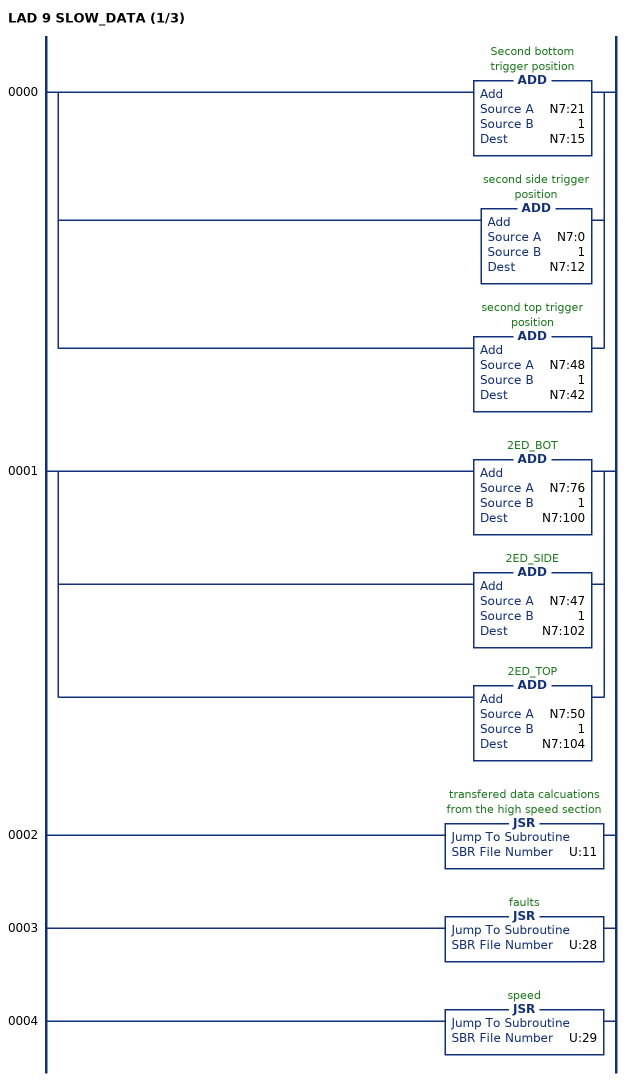
% Rung: 0 %
SOR BST ADD N7:21 1 N7:15 NXB ADD N7:0 1 N7:12 NXB ADD N7:48 1 N7:42 BND EOR
%   N7:21  BOT_TRIG_POS_INTEGER  "Trigger Position" %
%   N7:15  "Second bottom trigger position" %
%   N7:0  SIDE_TRIG_POS_INTEGE  "Side Trigger Position" %
%   N7:12  "second side trigger position" %
%   N7:48  TOP_TRIG_POS_INTEGER  "Top Trigger Position" %
%   N7:42  "second top trigger position" %
% Rung: 1 %
SOR BST ADD N7:76 1 N7:100 NXB ADD N7:47 1 N7:102 NXB ADD N7:50 1 N7:104 BND EOR
%   N7:76  BOT_TEST_LOC  "Location of pass window." %
%   N7:100  2ED_BOT %
%   N7:47  SIDE_TEST_LOC  "Location of pass window" %
%   N7:102  2ED_SIDE %
%   N7:50  TOP_TEST_LOC  "Location of pass window" %
%   N7:104  2ED_TOP %
% Rung: 2 %
SOR JSR U:11 EOR
%   U:11  "transfered data calcuations from the high speed section" %
% Rung: 3 %
SOR JSR U:28 EOR
%   U:28  "faults" %
% Rung: 4 %
SOR JSR U:29 EOR
%   U:29  "speed" %

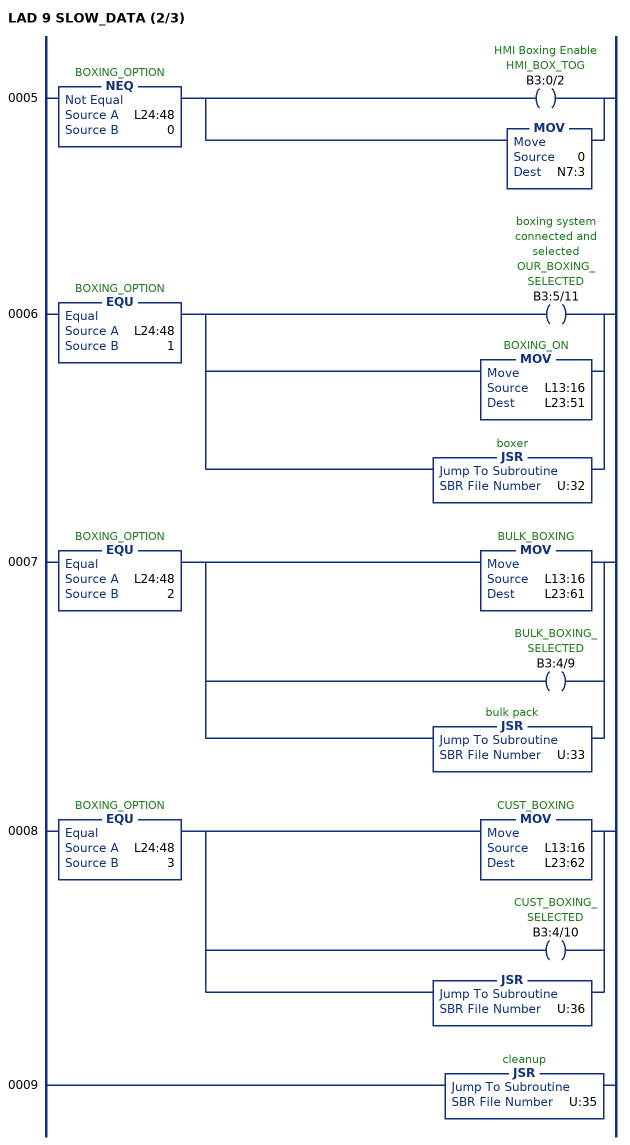
% Rung: 5 %
SOR NEQ L24:48 0 BST OTE B3:0/2 NXB MOV 0 N7:3 BND EOR
%   L24:48  BOXING_OPTION %
%   B3:0/2  HMI_BOX_TOG  "HMI Boxing Enable" %
% Rung: 6 %
SOR EQU L24:48 1 BST OTE B3:5/11 NXB MOV L13:16 L23:51 NXB JSR U:32 BND EOR
%   L24:48  BOXING_OPTION %
%   B3:5/11  OUR_BOXING_SELECTED  "boxing system connected and selected" %
%   L13:16  TRUE  "ONE TIME ENABLE FOR THE TIMES WHEN WE FORGET TO RE-ENABLE AFTER SHIPMENT" %
%   L23:51  BOXING_ON %
%   U:32  "boxer" %
% Rung: 7 %
SOR EQU L24:48 2 BST MOV L13:16 L23:61 NXB OTE B3:4/9 NXB JSR U:33 BND EOR
%   L24:48  BOXING_OPTION %
%   L13:16  TRUE  "ONE TIME ENABLE FOR THE TIMES WHEN WE FORGET TO RE-ENABLE AFTER SHIPMENT" %
%   L23:61  BULK_BOXING %
%   B3:4/9  BULK_BOXING_SELECTED %
%   U:33  "bulk pack" %
% Rung: 8 %
SOR EQU L24:48 3 BST MOV L13:16 L23:62 NXB OTE B3:4/10 NXB JSR U:36 BND EOR
%   L24:48  BOXING_OPTION %
%   L13:16  TRUE  "ONE TIME ENABLE FOR THE TIMES WHEN WE FORGET TO RE-ENABLE AFTER SHIPMENT" %
%   L23:62  CUST_BOXING %
%   B3:4/10  CUST_BOXING_SELECTED %
% Rung: 9 %
SOR JSR U:35 EOR
%   U:35  "cleanup" %

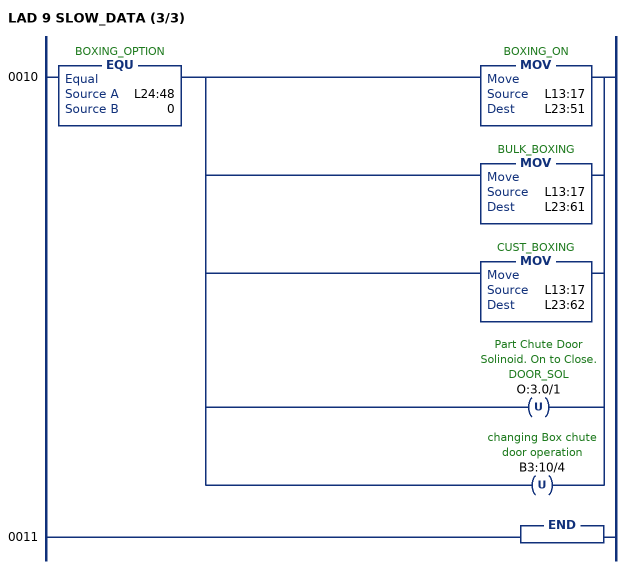
% Rung: 10 %
SOR EQU L24:48 0 BST MOV L13:17 L23:51 NXB MOV L13:17 L23:61 NXB MOV L13:17 L23:62 NXB OTU O:3.0/1 NXB OTU B3:10/4 BND EOR
%   L24:48  BOXING_OPTION %
%   L13:17  FALSE %
%   L23:51  BOXING_ON %
%   L23:61  BULK_BOXING %
%   L23:62  CUST_BOXING %
%   O:3.0/1  DOOR_SOL  "Part Chute Door Solinoid. On to Close." %
%   B3:10/4  "changing Box chute door operation" %
% Rung: 11 %
SOR END EOR

LADDER 10 "BOT_NUT"
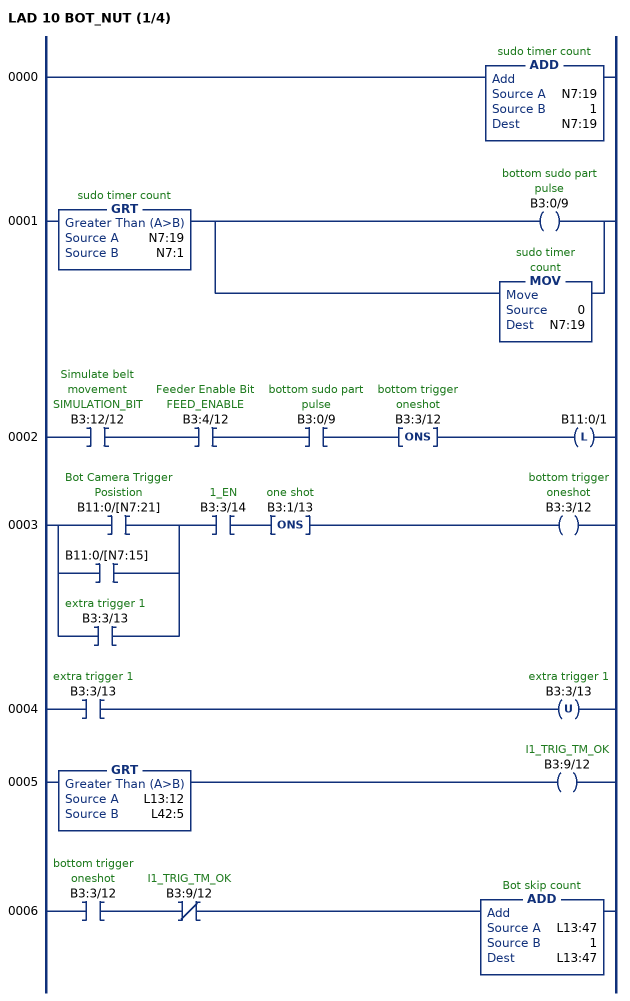
% Rung: 0 %
SOR ADD N7:19 1 N7:19 EOR
%   N7:19  "sudo timer count" %
% Rung: 1 %
SOR GRT N7:19 N7:1 BST OTE B3:0/9 NXB MOV 0 N7:19 BND EOR
%   N7:19  "sudo timer count" %
%   N7:1  "sudo part interval" %
%   B3:0/9  "bottom sudo part pulse" %
% Rung: 2 %
SOR XIC B3:12/12 XIC B3:4/12 XIC B3:0/9 ONS B3:3/12 OTL B11:0/1 EOR
%   B3:12/12  SIMULATION_BIT  "Simulate belt movement" %
%   B3:4/12  FEED_ENABLE  "Feeder Enable Bit" %
%   B3:0/9  "bottom sudo part pulse" %
%   B3:3/12  "bottom trigger oneshot" %
% Rung: 3 %
SOR BST XIC B11:0/[N7:21] NXB XIC B11:0/[N7:15] NXB XIC B3:3/13 BND XIC B3:3/14 ONS B3:1/13 OTE B3:3/12 EOR
%   B11:0/[N7:21]  "Bot Camera Trigger Posistion" %
%   N7:21  BOT_TRIG_POS_INTEGER  "Trigger Position" %
%   N7:15  "Second bottom trigger position" %
%   B3:3/13  "extra trigger 1" %
%   B3:3/14  1_EN %
%   B3:1/13  "one shot" %
%   B3:3/12  "bottom trigger oneshot" %
% Rung: 4 %
SOR XIC B3:3/13 OTU B3:3/13 EOR
%   B3:3/13  "extra trigger 1" %
% Rung: 5 %
SOR GRT L13:12 L42:5 OTE B3:9/12 EOR
%   B3:9/12  I1_TRIG_TM_OK %
% Rung: 6 %
SOR XIC B3:3/12 XIO B3:9/12 ADD L13:47 1 L13:47 EOR
%   B3:3/12  "bottom trigger oneshot" %
%   B3:9/12  I1_TRIG_TM_OK %
%   L13:47  "Bot skip count" %

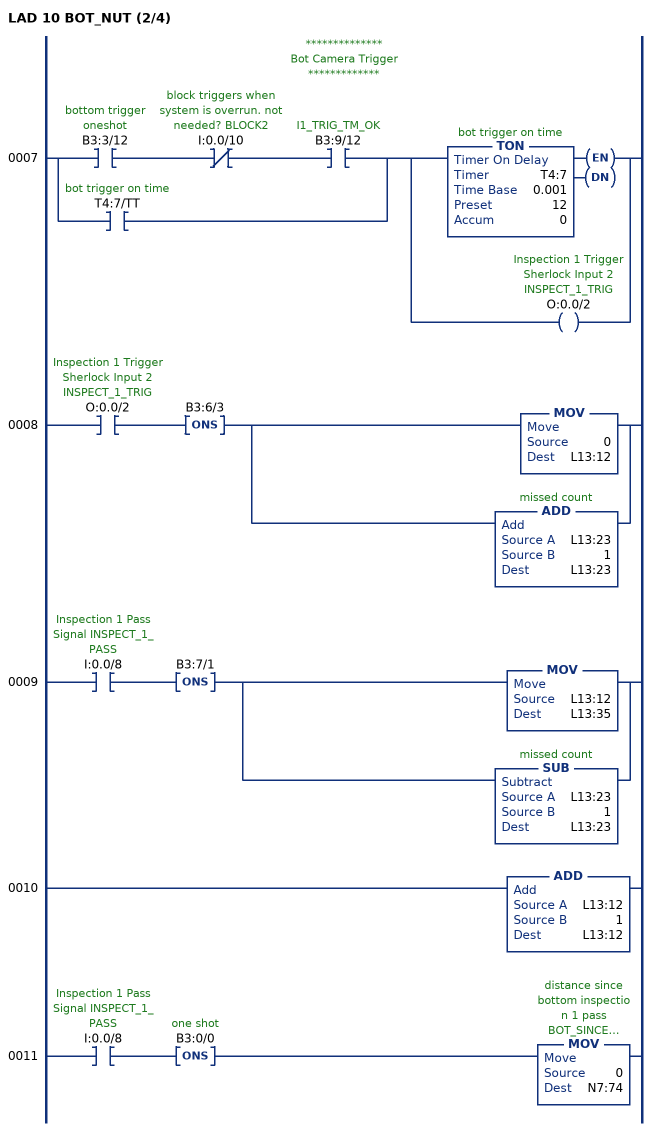
% Rung: 7 %
% **************
% Bot Camera Trigger
% ************* %
SOR BST XIC B3:3/12 XIO I:0.0/10 XIC B3:9/12 NXB XIC T4:7/TT BND BST TON T4:7 0.001 12 0 NXB OTE O:0.0/2 BND EOR
%   B3:3/12  "bottom trigger oneshot" %
%   I:0.0/10  BLOCK2  "block triggers when system is overrun. not needed?" %
%   B3:9/12  I1_TRIG_TM_OK %
%   T4:7  "bot trigger on time" %
%   O:0.0/2  INSPECT_1_TRIG  "Inspection 1 Trigger Sherlock Input 2" %
% Rung: 8 %
SOR XIC O:0.0/2 ONS B3:6/3 BST MOV 0 L13:12 NXB ADD L13:23 1 L13:23 BND EOR
%   O:0.0/2  INSPECT_1_TRIG  "Inspection 1 Trigger Sherlock Input 2" %
%   L13:23  "missed count" %
% Rung: 9 %
SOR XIC I:0.0/8 ONS B3:7/1 BST MOV L13:12 L13:35 NXB SUB L13:23 1 L13:23 BND EOR
%   I:0.0/8  INSPECT_1_PASS  "Inspection 1 Pass Signal" %
%   L13:23  "missed count" %
% Rung: 10 %
SOR ADD L13:12 1 L13:12 EOR
% Rung: 11 %
SOR XIC I:0.0/8 ONS B3:0/0 MOV 0 N7:74 EOR
%   I:0.0/8  INSPECT_1_PASS  "Inspection 1 Pass Signal" %
%   B3:0/0  "one shot" %
%   N7:74  BOT_SINCE_PASS  "distance since bottom inspection 1 pass" %

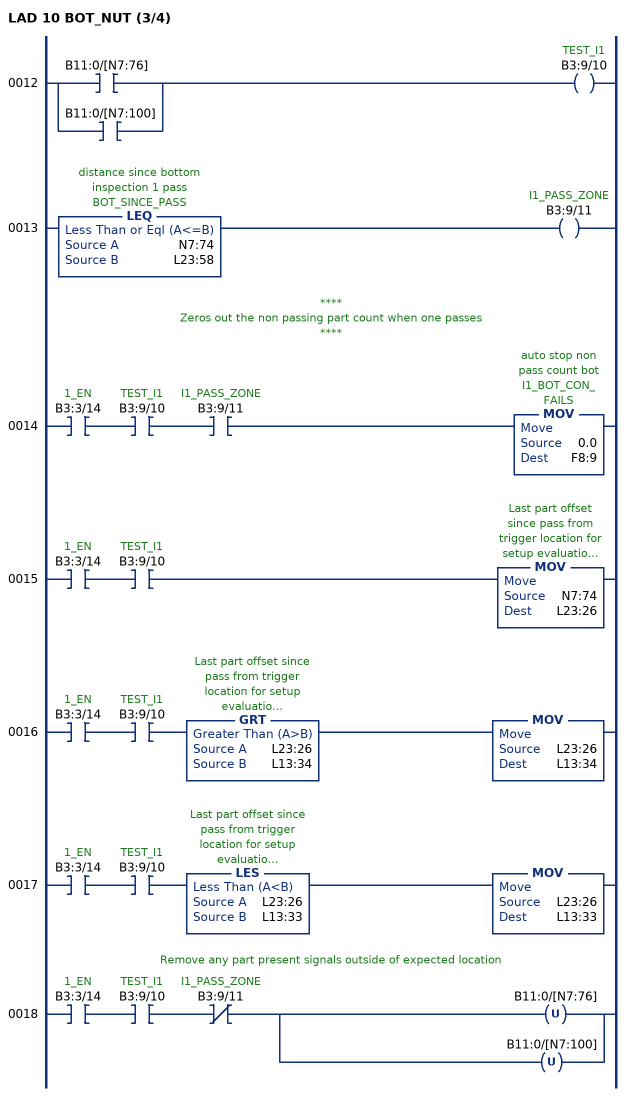
% Rung: 12 %
SOR BST XIC B11:0/[N7:76] NXB XIC B11:0/[N7:100] BND OTE B3:9/10 EOR
%   N7:76  BOT_TEST_LOC  "Location of pass window." %
%   N7:100  2ED_BOT %
%   B3:9/10  TEST_I1 %
% Rung: 13 %
SOR LEQ N7:74 L23:58 OTE B3:9/11 EOR
%   N7:74  BOT_SINCE_PASS  "distance since bottom inspection 1 pass" %
%   L23:58  BOT_RES_WIDTH %
%   B3:9/11  I1_PASS_ZONE %
% Rung: 14 %
% ****
%                   Zeros out the non passing part count when one passes
% **** %
SOR XIC B3:3/14 XIC B3:9/10 XIC B3:9/11 MOV 0.0 F8:9 EOR
%   B3:3/14  1_EN %
%   B3:9/10  TEST_I1 %
%   B3:9/11  I1_PASS_ZONE %
%   F8:9  I1_BOT_CON_FAILS  "auto stop non pass count bot" %
% Rung: 15 %
SOR XIC B3:3/14 XIC B3:9/10 MOV N7:74 L23:26 EOR
%   B3:3/14  1_EN %
%   B3:9/10  TEST_I1 %
%   N7:74  BOT_SINCE_PASS  "distance since bottom inspection 1 pass" %
%   L23:26  LAST_BOT_OFFSET  "Last part offset since pass from trigger location for setup evaluation" %
% Rung: 16 %
SOR XIC B3:3/14 XIC B3:9/10 GRT L23:26 L13:34 MOV L23:26 L13:34 EOR
%   B3:3/14  1_EN %
%   B3:9/10  TEST_I1 %
%   L23:26  LAST_BOT_OFFSET  "Last part offset since pass from trigger location for setup evaluation" %
% Rung: 17 %
SOR XIC B3:3/14 XIC B3:9/10 LES L23:26 L13:33 MOV L23:26 L13:33 EOR
%   B3:3/14  1_EN %
%   B3:9/10  TEST_I1 %
%   L23:26  LAST_BOT_OFFSET  "Last part offset since pass from trigger location for setup evaluation" %
% Rung: 18 %
% Remove any part present signals outside of expected location %
SOR XIC B3:3/14 XIC B3:9/10 XIO B3:9/11 BST OTU B11:0/[N7:76] NXB OTU B11:0/[N7:100] BND EOR
%   B3:3/14  1_EN %
%   B3:9/10  TEST_I1 %
%   B3:9/11  I1_PASS_ZONE %
%   N7:76  BOT_TEST_LOC  "Location of pass window." %
%   N7:100  2ED_BOT %

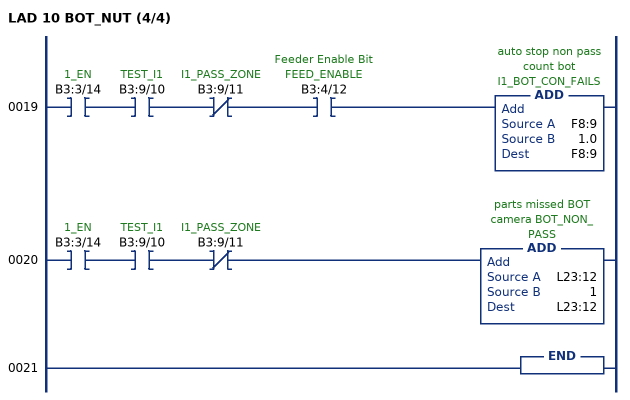
% Rung: 19 %
SOR XIC B3:3/14 XIC B3:9/10 XIO B3:9/11 XIC B3:4/12 ADD F8:9 1.0 F8:9 EOR
%   B3:3/14  1_EN %
%   B3:9/10  TEST_I1 %
%   B3:9/11  I1_PASS_ZONE %
%   B3:4/12  FEED_ENABLE  "Feeder Enable Bit" %
%   F8:9  I1_BOT_CON_FAILS  "auto stop non pass count bot" %
% Rung: 20 %
SOR XIC B3:3/14 XIC B3:9/10 XIO B3:9/11 ADD L23:12 1 L23:12 EOR
%   B3:3/14  1_EN %
%   B3:9/10  TEST_I1 %
%   B3:9/11  I1_PASS_ZONE %
%   L23:12  BOT_NON_PASS  "parts missed BOT camera" %
% Rung: 21 %
SOR END EOR

LADDER 11 "DATA_TRANS"
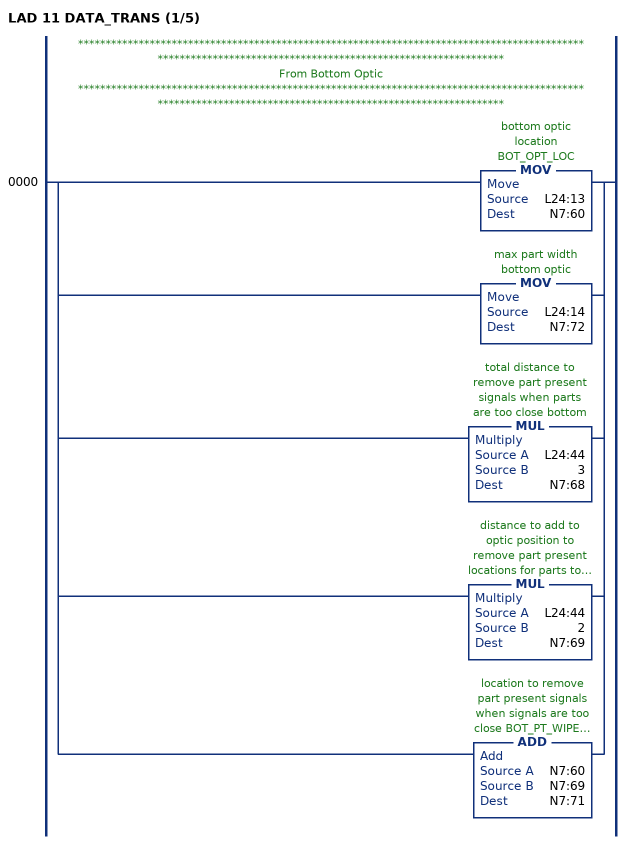
% Rung: 0 %
% ***********************************************************************************************************************************************************
% From Bottom Optic
% *********************************************************************************************************************************************************** %
SOR BST BST MOV L24:13 N7:60 NXB MOV L24:14 N7:72 BND NXB MUL L24:44 3 N7:68 NXB MUL L24:44 2 N7:69 NXB ADD N7:60 N7:69 N7:71 BND EOR
%   L24:13  BOT_OPTIC_LOC %
%   N7:60  BOT_OPT_LOC  "bottom optic location" %
%   L24:14  MAX_PART_WIDTH_BOT %
%   N7:72  "max part width bottom optic" %
%   L24:44  MIN_PART_GAP_BOT %
%   N7:68  "total distance to remove part present signals when parts are too close bottom" %
%   N7:69  "distance to add to optic position to remove part present locations for parts too close bottom" %
%   N7:71  BOT_PT_WIPE_LOC  "location to remove part present signals when signals are too close" %

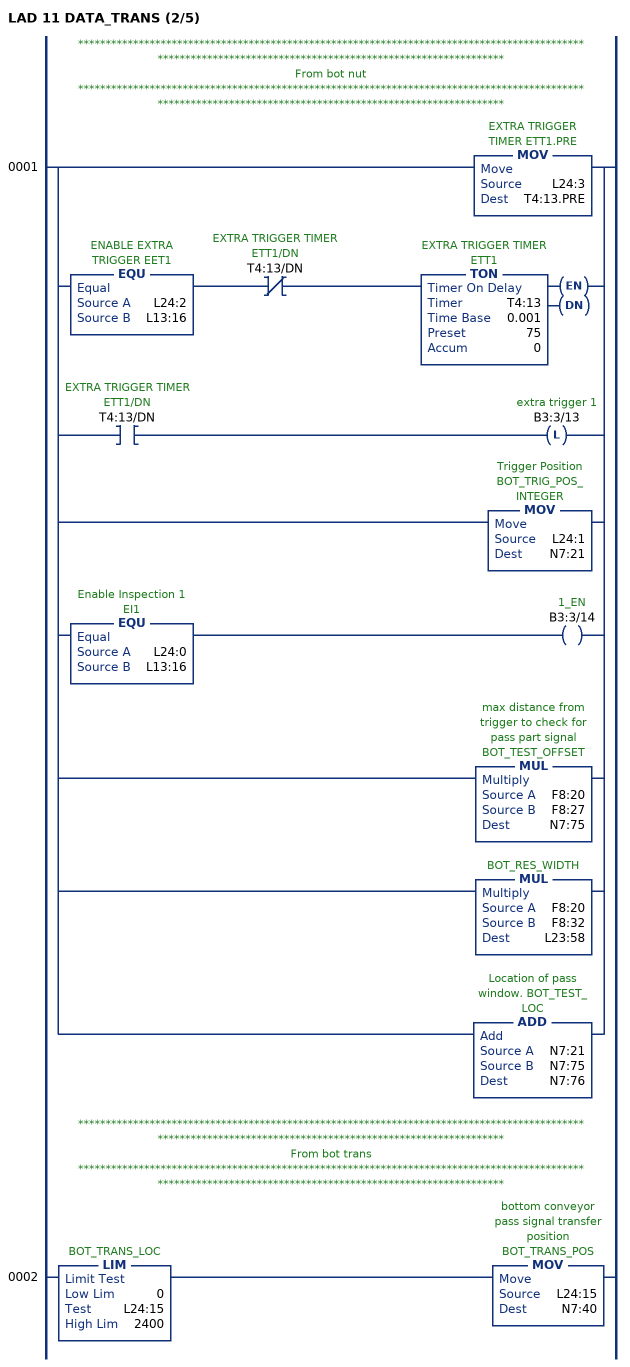
% Rung: 1 %
% ***********************************************************************************************************************************************************
% From bot nut
% *********************************************************************************************************************************************************** %
SOR BST BST MOV L24:3 T4:13.PRE NXB EQU L24:2 L13:16 XIO T4:13/DN TON T4:13 0.001 75 0 NXB XIC T4:13/DN OTL B3:3/13 NXB MOV L24:1 N7:21 NXB EQU L24:0 L13:16 OTE B3:3/14 BND NXB MUL F8:20 F8:27 N7:75 NXB MUL F8:20 F8:32 L23:58 NXB ADD N7:21 N7:75 N7:76 BND EOR
%   L24:3  ET1_DELAY %
%   T4:13  ETT1  "EXTRA TRIGGER TIMER" %
%   L24:2  EET1  "ENABLE EXTRA TRIGGER" %
%   L13:16  TRUE  "ONE TIME ENABLE FOR THE TIMES WHEN WE FORGET TO RE-ENABLE AFTER SHIPMENT" %
%   B3:3/13  "extra trigger 1" %
%   L24:1  I1_BOT_TRIG_LOC %
%   N7:21  BOT_TRIG_POS_INTEGER  "Trigger Position" %
%   L24:0  EI1  "Enable Inspection 1" %
%   B3:3/14  1_EN %
%   F8:20  "bot belt speed average in pulses per second" %
%   F8:27  MAX_TIME %
%   N7:75  BOT_TEST_OFFSET  "max distance from trigger to check for pass part signal" %
%   F8:32  TIME_WINDOW %
%   L23:58  BOT_RES_WIDTH %
%   N7:76  BOT_TEST_LOC  "Location of pass window." %
% Rung: 2 %
% ***********************************************************************************************************************************************************
% From bot trans
% *********************************************************************************************************************************************************** %
SOR LIM 0 L24:15 2400 MOV L24:15 N7:40 EOR
%   L24:15  BOT_TRANS_LOC %
%   N7:40  BOT_TRANS_POS  "bottom conveyor pass signal transfer position" %

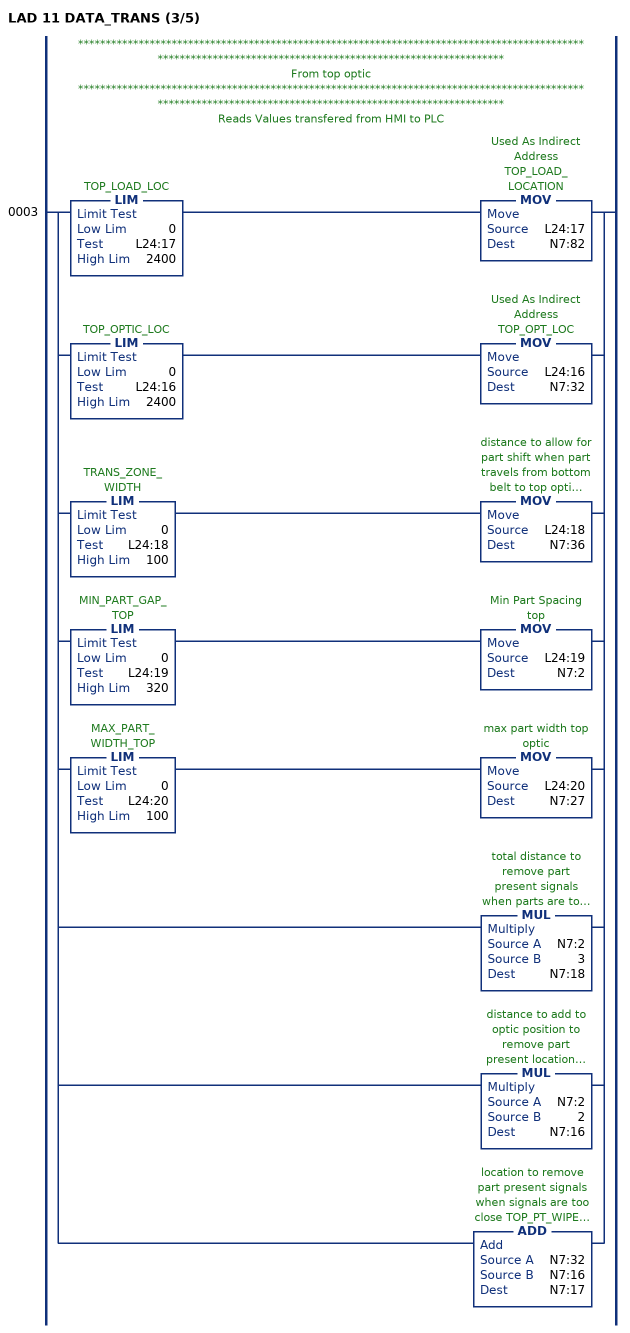
% Rung: 3 %
% ***********************************************************************************************************************************************************
% From top optic
% ***********************************************************************************************************************************************************
% 
% Reads Values transfered from HMI to PLC %
SOR BST BST LIM 0 L24:17 2400 MOV L24:17 N7:82 NXB LIM 0 L24:16 2400 MOV L24:16 N7:32 NXB LIM 0 L24:18 100 MOV L24:18 N7:36 NXB LIM 0 L24:19 320 MOV L24:19 N7:2 NXB LIM 0 L24:20 100 MOV L24:20 N7:27 BND NXB MUL N7:2 3 N7:18 NXB MUL N7:2 2 N7:16 NXB ADD N7:32 N7:16 N7:17 BND EOR
%   L24:17  TOP_LOAD_LOC %
%   N7:82  TOP_LOAD_LOCATION  "Used As Indirect Address" %
%   L24:16  TOP_OPTIC_LOC %
%   N7:32  TOP_OPT_LOC  "Used As Indirect Address" %
%   L24:18  TRANS_ZONE_WIDTH %
%   N7:36  TRANS_ZONE  "distance to allow for part shift when part travels from bottom belt to top optic" %
%   L24:19  MIN_PART_GAP_TOP %
%   N7:2  "Min Part Spacing top" %
%   L24:20  MAX_PART_WIDTH_TOP %
%   N7:27  "max part width top optic" %
%   N7:18  "total distance to remove part present signals when parts are too close top" %
%   N7:16  "distance to add to optic position to remove part present locations for parts too close top" %
%   N7:17  TOP_PT_WIPE_LOC  "location to remove part present signals when signals are too close" %

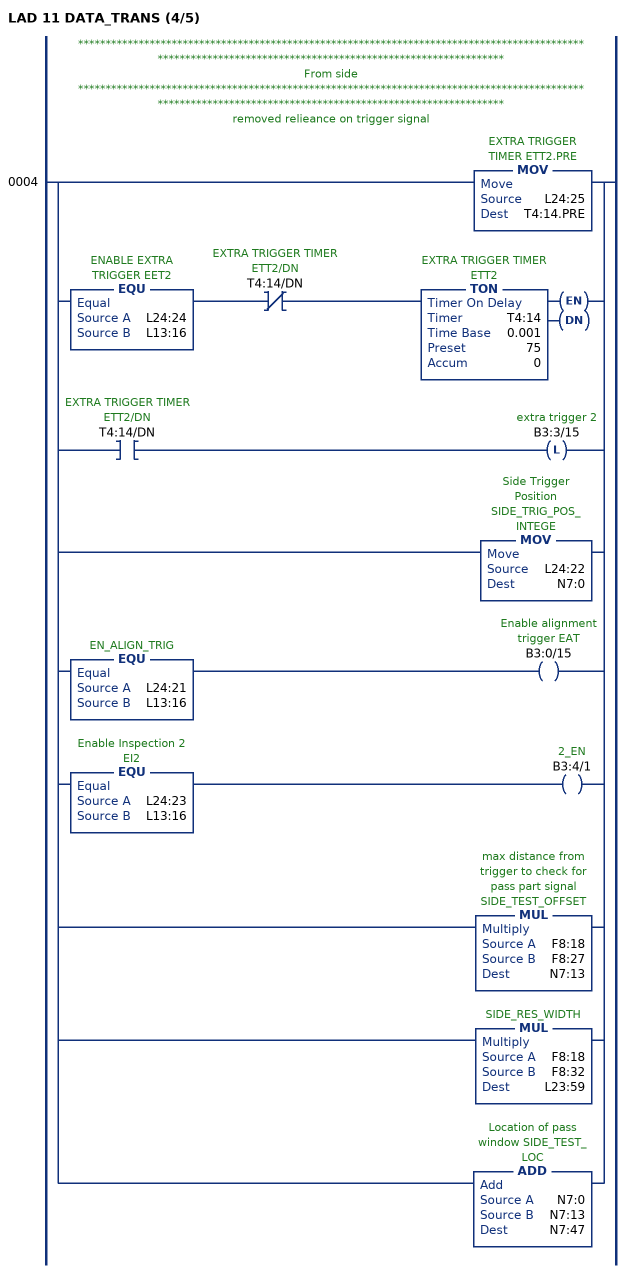
% Rung: 4 %
% ***********************************************************************************************************************************************************
% From side
% ***********************************************************************************************************************************************************
% 
% removed relieance on trigger signal %
SOR BST BST MOV L24:25 T4:14.PRE NXB EQU L24:24 L13:16 XIO T4:14/DN TON T4:14 0.001 75 0 NXB XIC T4:14/DN OTL B3:3/15 NXB MOV L24:22 N7:0 NXB EQU L24:21 L13:16 OTE B3:0/15 NXB EQU L24:23 L13:16 OTE B3:4/1 BND NXB MUL F8:18 F8:27 N7:13 NXB MUL F8:18 F8:32 L23:59 NXB ADD N7:0 N7:13 N7:47 BND EOR
%   L24:25  ET2_DELAY %
%   T4:14  ETT2  "EXTRA TRIGGER TIMER" %
%   L24:24  EET2  "ENABLE EXTRA TRIGGER" %
%   L13:16  TRUE  "ONE TIME ENABLE FOR THE TIMES WHEN WE FORGET TO RE-ENABLE AFTER SHIPMENT" %
%   B3:3/15  "extra trigger 2" %
%   L24:22  I2_SIDE_TRIG_LOC %
%   N7:0  SIDE_TRIG_POS_INTEGE  "Side Trigger Position" %
%   L24:21  EN_ALIGN_TRIG %
%   B3:0/15  EAT  "Enable alignment trigger" %
%   L24:23  EI2  "Enable Inspection 2" %
%   B3:4/1  2_EN %
%   F8:18  TOP_SPEED  "top belt speed average in pulses per second 290 Max; Verify" %
%   F8:27  MAX_TIME %
%   N7:13  SIDE_TEST_OFFSET  "max distance from trigger to check for pass part signal" %
%   F8:32  TIME_WINDOW %
%   L23:59  SIDE_RES_WIDTH %
%   N7:47  SIDE_TEST_LOC  "Location of pass window" %

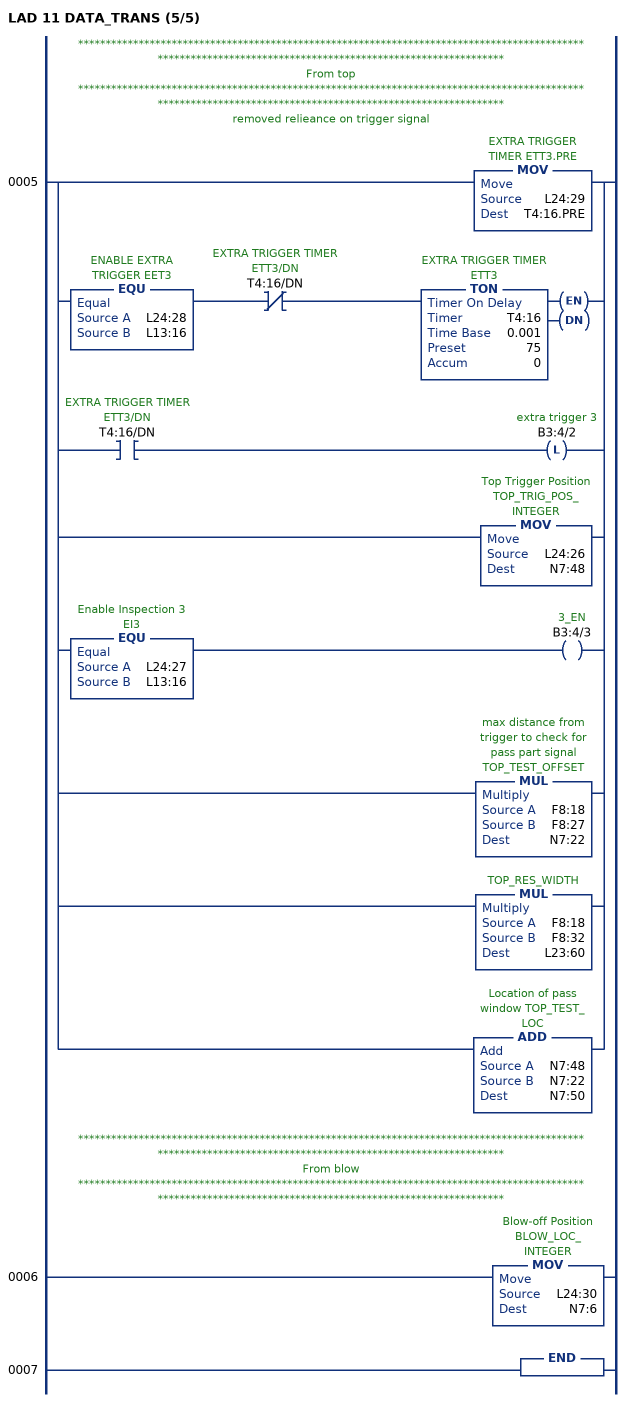
% Rung: 5 %
% ***********************************************************************************************************************************************************
% From top
% ***********************************************************************************************************************************************************
% 
% removed relieance on trigger signal %
SOR BST BST MOV L24:29 T4:16.PRE NXB EQU L24:28 L13:16 XIO T4:16/DN TON T4:16 0.001 75 0 NXB XIC T4:16/DN OTL B3:4/2 NXB MOV L24:26 N7:48 NXB EQU L24:27 L13:16 OTE B3:4/3 BND NXB MUL F8:18 F8:27 N7:22 NXB MUL F8:18 F8:32 L23:60 NXB ADD N7:48 N7:22 N7:50 BND EOR
%   L24:29  ET3_DELAY %
%   T4:16  ETT3  "EXTRA TRIGGER TIMER" %
%   L24:28  EET3  "ENABLE EXTRA TRIGGER" %
%   L13:16  TRUE  "ONE TIME ENABLE FOR THE TIMES WHEN WE FORGET TO RE-ENABLE AFTER SHIPMENT" %
%   B3:4/2  "extra trigger 3" %
%   L24:26  I3_TOP_TRIG_LOC %
%   N7:48  TOP_TRIG_POS_INTEGER  "Top Trigger Position" %
%   L24:27  EI3  "Enable Inspection 3" %
%   B3:4/3  3_EN %
%   F8:18  TOP_SPEED  "top belt speed average in pulses per second 290 Max; Verify" %
%   F8:27  MAX_TIME %
%   N7:22  TOP_TEST_OFFSET  "max distance from trigger to check for pass part signal" %
%   F8:32  TIME_WINDOW %
%   L23:60  TOP_RES_WIDTH %
%   N7:50  TOP_TEST_LOC  "Location of pass window" %
% Rung: 6 %
% ***********************************************************************************************************************************************************
% From blow
% *********************************************************************************************************************************************************** %
SOR MOV L24:30 N7:6 EOR
%   L24:30  BLOW_OFF_LOC %
%   N7:6  BLOW_LOC_INTEGER  "Blow-off Position" %
% Rung: 7 %
SOR END EOR

LADDER 12 "BOT_TRANSF"
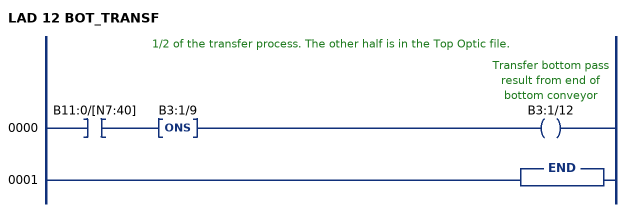
% Rung: 0 %
% 1/2 of the transfer process. The other half is in the Top Optic file. %
SOR XIC B11:0/[N7:40] ONS B3:1/9 OTE B3:1/12 EOR
%   N7:40  BOT_TRANS_POS  "bottom conveyor pass signal transfer position" %
%   B3:1/12  "Transfer bottom pass result from end of bottom conveyor" %
% Rung: 1 %
SOR END EOR

LADDER 14 "TOP_OPTIC"
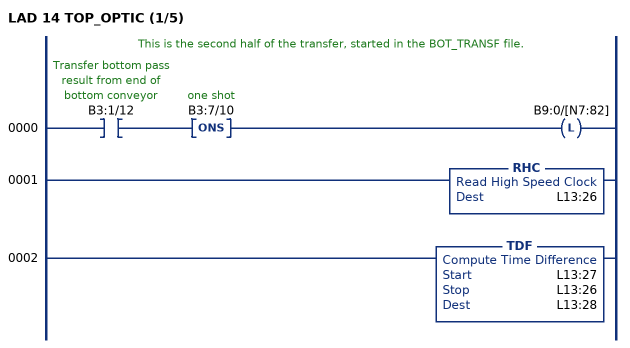
% Rung: 0 %
% This is the second half of the transfer, started in the BOT_TRANSF file. %
SOR XIC B3:1/12 ONS B3:7/10 OTL B9:0/[N7:82] EOR
%   B3:1/12  "Transfer bottom pass result from end of bottom conveyor" %
%   B3:7/10  "one shot" %
%   N7:82  TOP_LOAD_LOCATION  "Used As Indirect Address" %
% Rung: 1 %
SOR RHC L13:26 EOR
% Rung: 2 %
SOR TDF L13:27 L13:26 L13:28 EOR

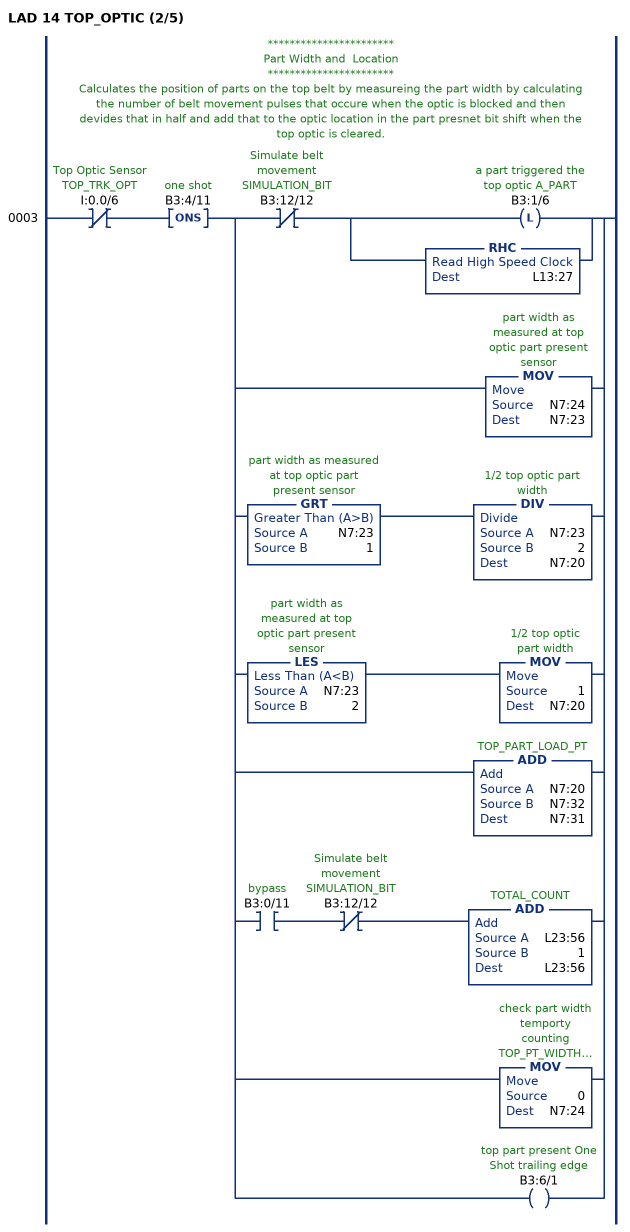
% Rung: 3 %
% ***********************
% Part Width and  Location
% ***********************
% 
% Calculates the position of parts on the top belt by measureing the part width by calculating the number of belt movement pulses that occure when the optic is blocked and then devides that in half and add that to the optic location in the part presnet bit shift when the top optic is cleared. %
SOR XIO I:0.0/6 ONS B3:4/11 BST XIO B3:12/12 BST OTL B3:1/6 NXB RHC L13:27 BND NXB MOV N7:24 N7:23 NXB GRT N7:23 1 DIV N7:23 2 N7:20 NXB LES N7:23 2 MOV 1 N7:20 NXB ADD N7:20 N7:32 N7:31 NXB XIC B3:0/11 XIO B3:12/12 ADD L23:56 1 L23:56 NXB MOV 0 N7:24 NXB OTE B3:6/1 BND EOR
%   I:0.0/6  TOP_TRK_OPT  "Top Optic Sensor" %
%   B3:4/11  "one shot" %
%   B3:12/12  SIMULATION_BIT  "Simulate belt movement" %
%   B3:1/6  A_PART  "a part triggered the top optic" %
%   N7:24  TOP_PT_WIDTH_TEMP  "check part width temporty counting" %
%   N7:23  "part width as measured at top optic part present sensor" %
%   N7:20  "1/2 top optic part width" %
%   N7:32  TOP_OPT_LOC  "Used As Indirect Address" %
%   N7:31  TOP_PART_LOAD_PT %
%   B3:0/11  "bypass" %
%   L23:56  TOTAL_COUNT %
%   B3:6/1  "top part present One Shot trailing edge" %

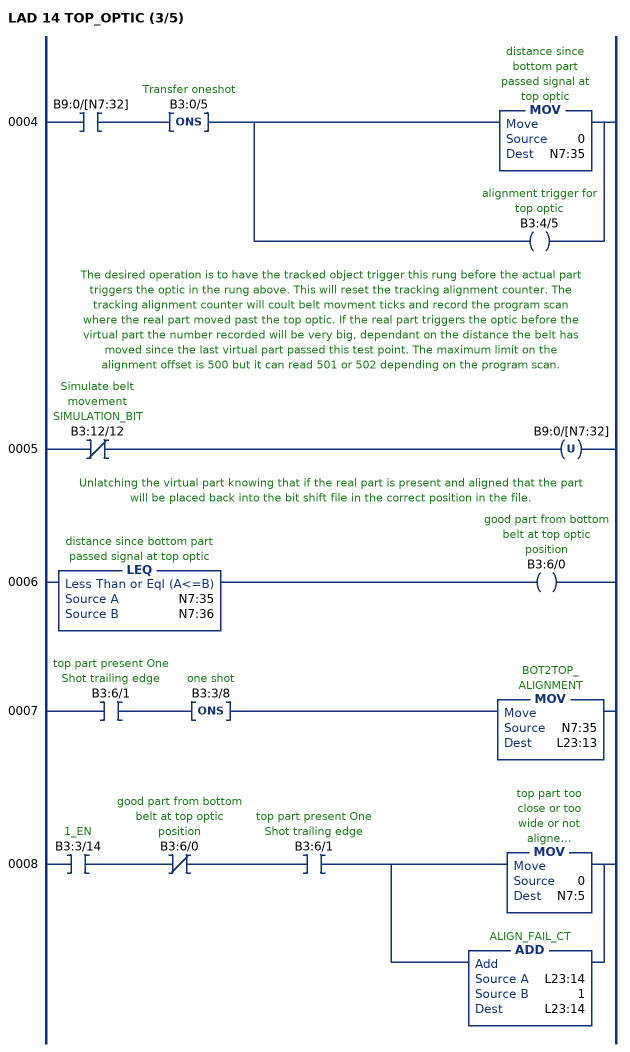
% Rung: 4 %
SOR XIC B9:0/[N7:32] ONS B3:0/5 BST MOV 0 N7:35 NXB OTE B3:4/5 BND EOR
%   N7:32  TOP_OPT_LOC  "Used As Indirect Address" %
%   B3:0/5  "Transfer oneshot" %
%   N7:35  "distance since bottom part passed signal at top optic" %
%   B3:4/5  "alignment trigger for top optic" %
% Rung: 5 %
% The desired operation is to have the tracked object trigger this rung before the actual part triggers the optic in the rung above. This will reset the tracking alignment counter. The tracking alignment counter will coult belt movment ticks and record the program scan where the real part moved past the top optic. If the real part triggers the optic before the virtual part the number recorded will be very big, dependant on the distance the belt has moved since the last virtual part passed this test point. The maximum limit on the alignment offset is 500 but it can read 501 or 502 depending on the program scan. %
SOR XIO B3:12/12 OTU B9:0/[N7:32] EOR
%   B3:12/12  SIMULATION_BIT  "Simulate belt movement" %
%   N7:32  TOP_OPT_LOC  "Used As Indirect Address" %
% Rung: 6 %
% Unlatching the virtual part knowing that if the real part is present and aligned that the part will be placed back into the bit shift file in the correct position in the file. %
SOR LEQ N7:35 N7:36 OTE B3:6/0 EOR
%   N7:35  "distance since bottom part passed signal at top optic" %
%   N7:36  TRANS_ZONE  "distance to allow for part shift when part travels from bottom belt to top optic" %
%   B3:6/0  "good part from bottom belt at top optic position" %
% Rung: 7 %
SOR XIC B3:6/1 ONS B3:3/8 MOV N7:35 L23:13 EOR
%   B3:6/1  "top part present One Shot trailing edge" %
%   B3:3/8  "one shot" %
%   N7:35  "distance since bottom part passed signal at top optic" %
%   L23:13  BOT2TOP_ALIGNMENT %
% Rung: 8 %
SOR XIC B3:3/14 XIO B3:6/0 XIC B3:6/1 BST MOV 0 N7:5 NXB ADD L23:14 1 L23:14 BND EOR
%   B3:3/14  1_EN %
%   B3:6/0  "good part from bottom belt at top optic position" %
%   B3:6/1  "top part present One Shot trailing edge" %
%   N7:5  "top part too close or too wide or not aligned distance measurement" %
%   L23:14  ALIGN_FAIL_CT %

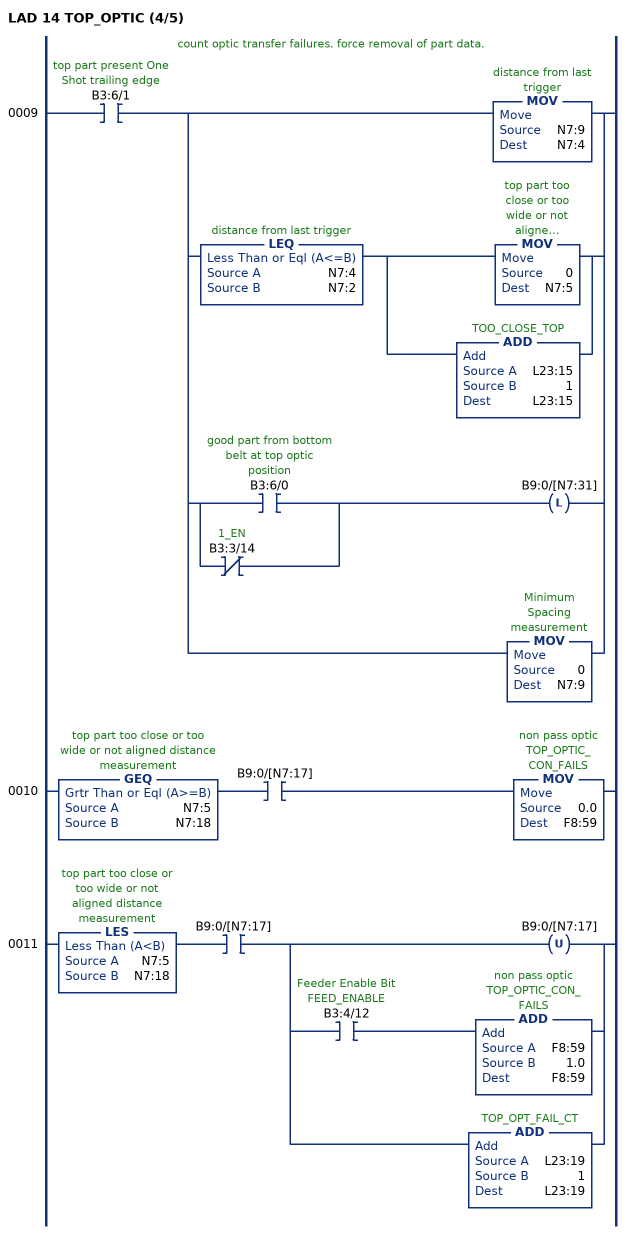
% Rung: 9 %
% count optic transfer failures. force removal of part data. %
SOR XIC B3:6/1 BST MOV N7:9 N7:4 NXB LEQ N7:4 N7:2 BST MOV 0 N7:5 NXB ADD L23:15 1 L23:15 BND NXB BST XIC B3:6/0 NXB XIO B3:3/14 BND OTL B9:0/[N7:31] NXB MOV 0 N7:9 BND EOR
%   B3:6/1  "top part present One Shot trailing edge" %
%   N7:9  "Minimum Spacing measurement" %
%   N7:4  "distance from last trigger" %
%   N7:2  "Min Part Spacing top" %
%   N7:5  "top part too close or too wide or not aligned distance measurement" %
%   L23:15  TOO_CLOSE_TOP %
%   B3:6/0  "good part from bottom belt at top optic position" %
%   B3:3/14  1_EN %
%   N7:31  TOP_PART_LOAD_PT %
% Rung: 10 %
SOR GEQ N7:5 N7:18 XIC B9:0/[N7:17] MOV 0.0 F8:59 EOR
%   N7:5  "top part too close or too wide or not aligned distance measurement" %
%   N7:18  "total distance to remove part present signals when parts are too close top" %
%   N7:17  TOP_PT_WIPE_LOC  "location to remove part present signals when signals are too close" %
%   F8:59  TOP_OPTIC_CON_FAILS  "non pass optic" %
% Rung: 11 %
SOR LES N7:5 N7:18 XIC B9:0/[N7:17] BST OTU B9:0/[N7:17] NXB XIC B3:4/12 ADD F8:59 1.0 F8:59 NXB ADD L23:19 1 L23:19 BND EOR
%   N7:5  "top part too close or too wide or not aligned distance measurement" %
%   N7:18  "total distance to remove part present signals when parts are too close top" %
%   N7:17  TOP_PT_WIPE_LOC  "location to remove part present signals when signals are too close" %
%   B3:4/12  FEED_ENABLE  "Feeder Enable Bit" %
%   F8:59  TOP_OPTIC_CON_FAILS  "non pass optic" %
%   L23:19  TOP_OPT_FAIL_CT %

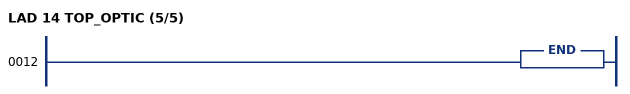
% Rung: 12 %
SOR END EOR

LADDER 16 "TOP_SIDE"
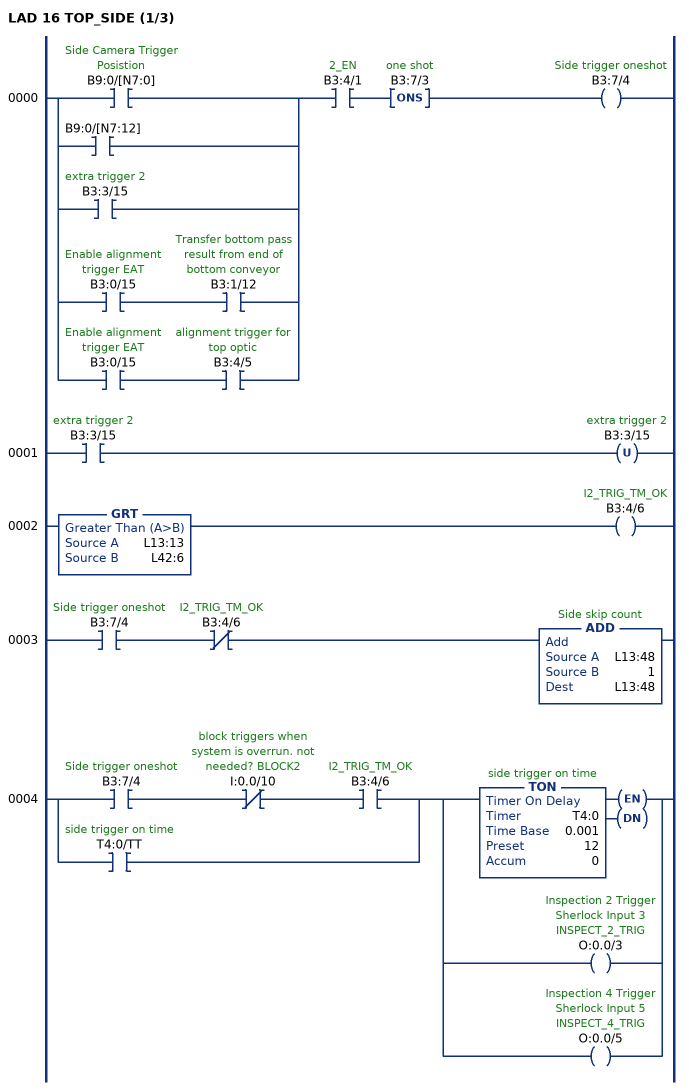
% Rung: 0 %
SOR BST XIC B9:0/[N7:0] NXB XIC B9:0/[N7:12] NXB XIC B3:3/15 NXB XIC B3:0/15 XIC B3:1/12 NXB XIC B3:0/15 XIC B3:4/5 BND XIC B3:4/1 ONS B3:7/3 OTE B3:7/4 EOR
%   B9:0/[N7:0]  "Side Camera Trigger Posistion" %
%   N7:0  SIDE_TRIG_POS_INTEGE  "Side Trigger Position" %
%   N7:12  "second side trigger position" %
%   B3:3/15  "extra trigger 2" %
%   B3:0/15  EAT  "Enable alignment trigger" %
%   B3:1/12  "Transfer bottom pass result from end of bottom conveyor" %
%   B3:4/5  "alignment trigger for top optic" %
%   B3:4/1  2_EN %
%   B3:7/3  "one shot" %
%   B3:7/4  "Side trigger oneshot" %
% Rung: 1 %
SOR XIC B3:3/15 OTU B3:3/15 EOR
%   B3:3/15  "extra trigger 2" %
% Rung: 2 %
SOR GRT L13:13 L42:6 OTE B3:4/6 EOR
%   B3:4/6  I2_TRIG_TM_OK %
% Rung: 3 %
SOR XIC B3:7/4 XIO B3:4/6 ADD L13:48 1 L13:48 EOR
%   B3:7/4  "Side trigger oneshot" %
%   B3:4/6  I2_TRIG_TM_OK %
%   L13:48  "Side skip count" %
% Rung: 4 %
SOR BST XIC B3:7/4 XIO I:0.0/10 XIC B3:4/6 NXB XIC T4:0/TT BND BST TON T4:0 0.001 12 0 NXB OTE O:0.0/3 NXB OTE O:0.0/5 BND EOR
%   B3:7/4  "Side trigger oneshot" %
%   I:0.0/10  BLOCK2  "block triggers when system is overrun. not needed?" %
%   B3:4/6  I2_TRIG_TM_OK %
%   T4:0  "side trigger on time" %
%   O:0.0/3  INSPECT_2_TRIG  "Inspection 2 Trigger Sherlock Input 3" %
%   O:0.0/5  INSPECT_4_TRIG  "Inspection 4 Trigger Sherlock Input 5" %

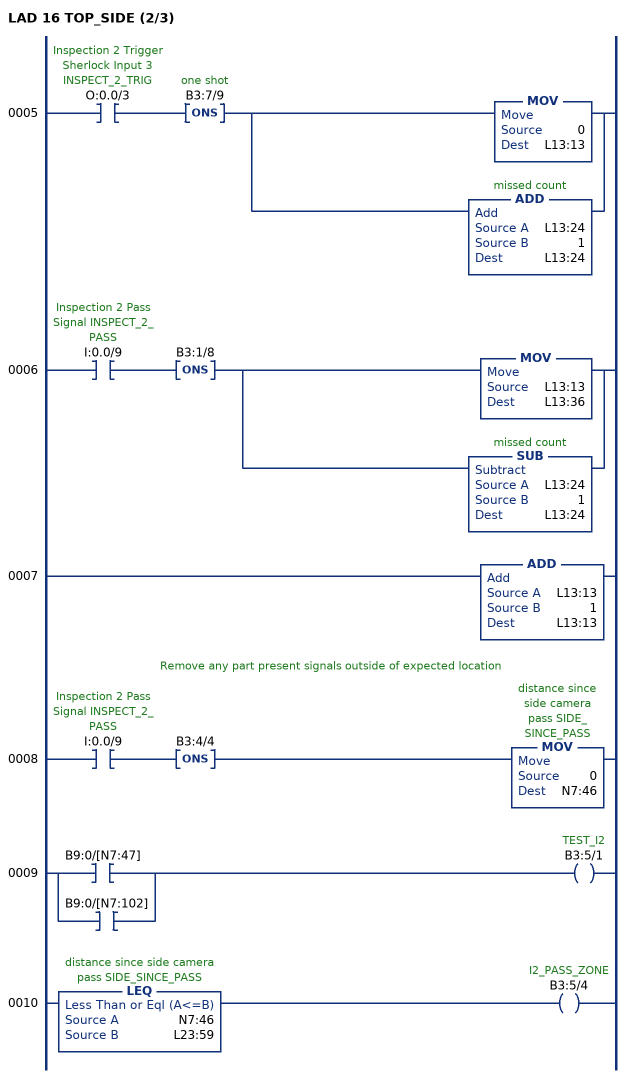
% Rung: 5 %
SOR XIC O:0.0/3 ONS B3:7/9 BST MOV 0 L13:13 NXB ADD L13:24 1 L13:24 BND EOR
%   O:0.0/3  INSPECT_2_TRIG  "Inspection 2 Trigger Sherlock Input 3" %
%   B3:7/9  "one shot" %
%   L13:24  "missed count" %
% Rung: 6 %
SOR XIC I:0.0/9 ONS B3:1/8 BST MOV L13:13 L13:36 NXB SUB L13:24 1 L13:24 BND EOR
%   I:0.0/9  INSPECT_2_PASS  "Inspection 2 Pass Signal" %
%   L13:24  "missed count" %
% Rung: 7 %
SOR ADD L13:13 1 L13:13 EOR
% Rung: 8 %
% Remove any part present signals outside of expected location %
SOR XIC I:0.0/9 ONS B3:4/4 MOV 0 N7:46 EOR
%   I:0.0/9  INSPECT_2_PASS  "Inspection 2 Pass Signal" %
%   N7:46  SIDE_SINCE_PASS  "distance since side camera pass" %
% Rung: 9 %
SOR BST XIC B9:0/[N7:47] NXB XIC B9:0/[N7:102] BND OTE B3:5/1 EOR
%   N7:47  SIDE_TEST_LOC  "Location of pass window" %
%   N7:102  2ED_SIDE %
%   B3:5/1  TEST_I2 %
% Rung: 10 %
SOR LEQ N7:46 L23:59 OTE B3:5/4 EOR
%   N7:46  SIDE_SINCE_PASS  "distance since side camera pass" %
%   L23:59  SIDE_RES_WIDTH %
%   B3:5/4  I2_PASS_ZONE %

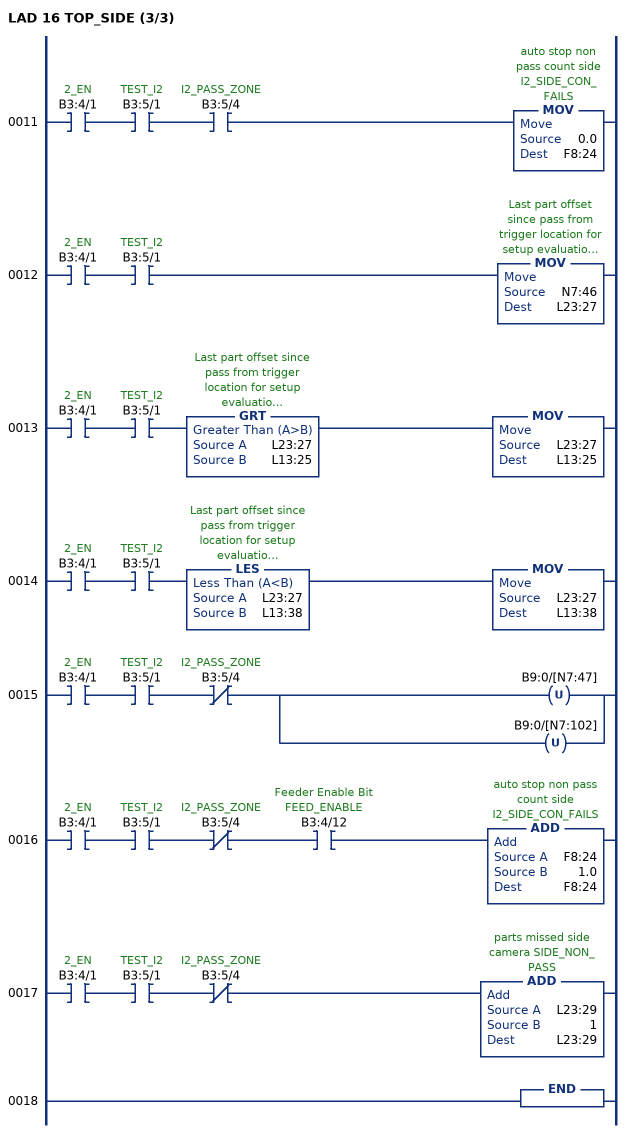
% Rung: 11 %
SOR XIC B3:4/1 XIC B3:5/1 XIC B3:5/4 MOV 0.0 F8:24 EOR
%   B3:4/1  2_EN %
%   B3:5/1  TEST_I2 %
%   B3:5/4  I2_PASS_ZONE %
%   F8:24  I2_SIDE_CON_FAILS  "auto stop non pass count side" %
% Rung: 12 %
SOR XIC B3:4/1 XIC B3:5/1 MOV N7:46 L23:27 EOR
%   B3:4/1  2_EN %
%   B3:5/1  TEST_I2 %
%   N7:46  SIDE_SINCE_PASS  "distance since side camera pass" %
%   L23:27  LAST_SIDE_OFFSET  "Last part offset since pass from trigger location for setup evaluation" %
% Rung: 13 %
SOR XIC B3:4/1 XIC B3:5/1 GRT L23:27 L13:25 MOV L23:27 L13:25 EOR
%   B3:4/1  2_EN %
%   B3:5/1  TEST_I2 %
%   L23:27  LAST_SIDE_OFFSET  "Last part offset since pass from trigger location for setup evaluation" %
% Rung: 14 %
SOR XIC B3:4/1 XIC B3:5/1 LES L23:27 L13:38 MOV L23:27 L13:38 EOR
%   B3:4/1  2_EN %
%   B3:5/1  TEST_I2 %
%   L23:27  LAST_SIDE_OFFSET  "Last part offset since pass from trigger location for setup evaluation" %
% Rung: 15 %
SOR XIC B3:4/1 XIC B3:5/1 XIO B3:5/4 BST OTU B9:0/[N7:47] NXB OTU B9:0/[N7:102] BND EOR
%   B3:4/1  2_EN %
%   B3:5/1  TEST_I2 %
%   B3:5/4  I2_PASS_ZONE %
%   N7:47  SIDE_TEST_LOC  "Location of pass window" %
%   N7:102  2ED_SIDE %
% Rung: 16 %
SOR XIC B3:4/1 XIC B3:5/1 XIO B3:5/4 XIC B3:4/12 ADD F8:24 1.0 F8:24 EOR
%   B3:4/1  2_EN %
%   B3:5/1  TEST_I2 %
%   B3:5/4  I2_PASS_ZONE %
%   B3:4/12  FEED_ENABLE  "Feeder Enable Bit" %
%   F8:24  I2_SIDE_CON_FAILS  "auto stop non pass count side" %
% Rung: 17 %
SOR XIC B3:4/1 XIC B3:5/1 XIO B3:5/4 ADD L23:29 1 L23:29 EOR
%   B3:4/1  2_EN %
%   B3:5/1  TEST_I2 %
%   B3:5/4  I2_PASS_ZONE %
%   L23:29  SIDE_NON_PASS  "parts missed side camera" %
% Rung: 18 %
SOR END EOR

LADDER 20 "TOP_TOP"
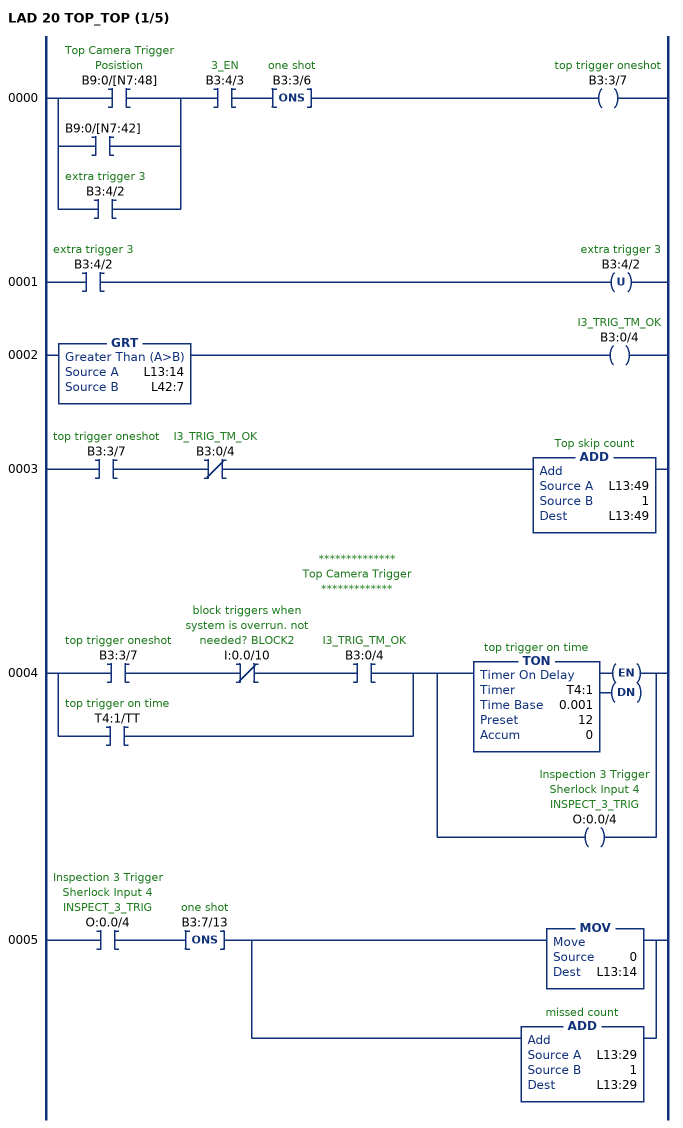
% Rung: 0 %
SOR BST XIC B9:0/[N7:48] NXB XIC B9:0/[N7:42] NXB XIC B3:4/2 BND XIC B3:4/3 ONS B3:3/6 OTE B3:3/7 EOR
%   B9:0/[N7:48]  "Top Camera Trigger Posistion" %
%   N7:48  TOP_TRIG_POS_INTEGER  "Top Trigger Position" %
%   N7:42  "second top trigger position" %
%   B3:4/2  "extra trigger 3" %
%   B3:4/3  3_EN %
%   B3:3/6  "one shot" %
%   B3:3/7  "top trigger oneshot" %
% Rung: 1 %
SOR XIC B3:4/2 OTU B3:4/2 EOR
%   B3:4/2  "extra trigger 3" %
% Rung: 2 %
SOR GRT L13:14 L42:7 OTE B3:0/4 EOR
%   B3:0/4  I3_TRIG_TM_OK %
% Rung: 3 %
SOR XIC B3:3/7 XIO B3:0/4 ADD L13:49 1 L13:49 EOR
%   B3:3/7  "top trigger oneshot" %
%   B3:0/4  I3_TRIG_TM_OK %
%   L13:49  "Top skip count" %
% Rung: 4 %
% **************
% Top Camera Trigger
% ************* %
SOR BST XIC B3:3/7 XIO I:0.0/10 XIC B3:0/4 NXB XIC T4:1/TT BND BST TON T4:1 0.001 12 0 NXB OTE O:0.0/4 BND EOR
%   B3:3/7  "top trigger oneshot" %
%   I:0.0/10  BLOCK2  "block triggers when system is overrun. not needed?" %
%   B3:0/4  I3_TRIG_TM_OK %
%   T4:1  "top trigger on time" %
%   O:0.0/4  INSPECT_3_TRIG  "Inspection 3 Trigger Sherlock Input 4" %
% Rung: 5 %
SOR XIC O:0.0/4 ONS B3:7/13 BST MOV 0 L13:14 NXB ADD L13:29 1 L13:29 BND EOR
%   O:0.0/4  INSPECT_3_TRIG  "Inspection 3 Trigger Sherlock Input 4" %
%   B3:7/13  "one shot" %
%   L13:29  "missed count" %

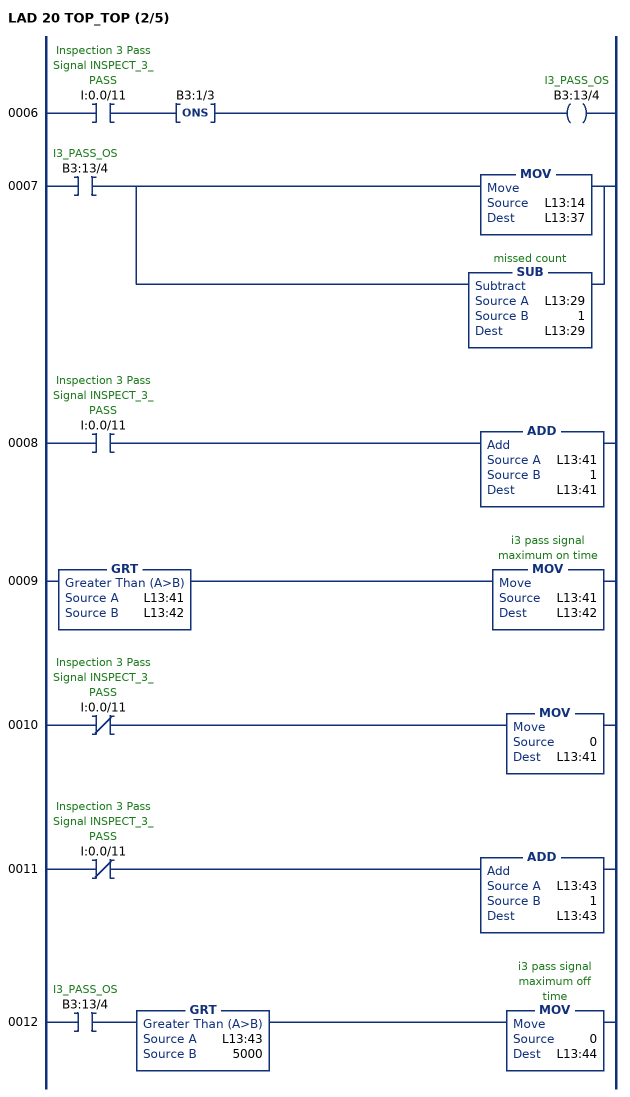
% Rung: 6 %
SOR XIC I:0.0/11 ONS B3:1/3 OTE B3:13/4 EOR
%   I:0.0/11  INSPECT_3_PASS  "Inspection 3 Pass Signal" %
%   B3:13/4  I3_PASS_OS %
% Rung: 7 %
SOR XIC B3:13/4 BST MOV L13:14 L13:37 NXB SUB L13:29 1 L13:29 BND EOR
%   B3:13/4  I3_PASS_OS %
%   L13:29  "missed count" %
% Rung: 8 %
SOR XIC I:0.0/11 ADD L13:41 1 L13:41 EOR
%   I:0.0/11  INSPECT_3_PASS  "Inspection 3 Pass Signal" %
% Rung: 9 %
SOR GRT L13:41 L13:42 MOV L13:41 L13:42 EOR
%   L13:42  "i3 pass signal maximum on time" %
% Rung: 10 %
SOR XIO I:0.0/11 MOV 0 L13:41 EOR
%   I:0.0/11  INSPECT_3_PASS  "Inspection 3 Pass Signal" %
% Rung: 11 %
SOR XIO I:0.0/11 ADD L13:43 1 L13:43 EOR
%   I:0.0/11  INSPECT_3_PASS  "Inspection 3 Pass Signal" %
% Rung: 12 %
SOR XIC B3:13/4 GRT L13:43 5000 MOV 0 L13:44 EOR
%   B3:13/4  I3_PASS_OS %
%   L13:44  "i3 pass signal maximum off time" %

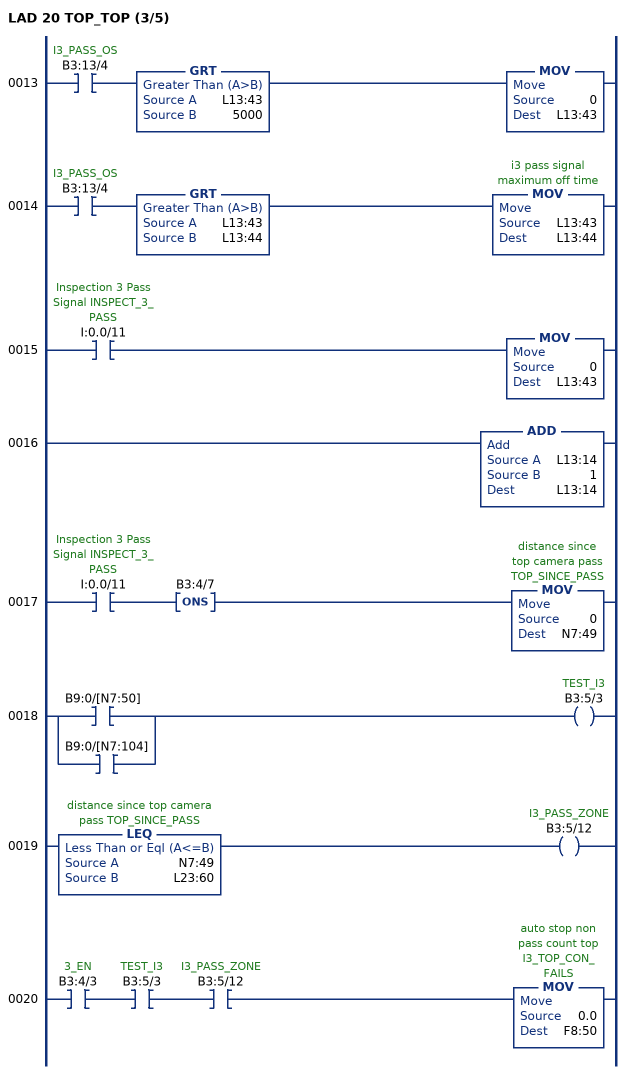
% Rung: 13 %
SOR XIC B3:13/4 GRT L13:43 5000 MOV 0 L13:43 EOR
%   B3:13/4  I3_PASS_OS %
% Rung: 14 %
SOR XIC B3:13/4 GRT L13:43 L13:44 MOV L13:43 L13:44 EOR
%   B3:13/4  I3_PASS_OS %
%   L13:44  "i3 pass signal maximum off time" %
% Rung: 15 %
SOR XIC I:0.0/11 MOV 0 L13:43 EOR
%   I:0.0/11  INSPECT_3_PASS  "Inspection 3 Pass Signal" %
% Rung: 16 %
SOR ADD L13:14 1 L13:14 EOR
% Rung: 17 %
SOR XIC I:0.0/11 ONS B3:4/7 MOV 0 N7:49 EOR
%   I:0.0/11  INSPECT_3_PASS  "Inspection 3 Pass Signal" %
%   N7:49  TOP_SINCE_PASS  "distance since top camera pass" %
% Rung: 18 %
SOR BST XIC B9:0/[N7:50] NXB XIC B9:0/[N7:104] BND OTE B3:5/3 EOR
%   N7:50  TOP_TEST_LOC  "Location of pass window" %
%   N7:104  2ED_TOP %
%   B3:5/3  TEST_I3 %
% Rung: 19 %
SOR LEQ N7:49 L23:60 OTE B3:5/12 EOR
%   N7:49  TOP_SINCE_PASS  "distance since top camera pass" %
%   L23:60  TOP_RES_WIDTH %
%   B3:5/12  I3_PASS_ZONE %
% Rung: 20 %
SOR XIC B3:4/3 XIC B3:5/3 XIC B3:5/12 MOV 0.0 F8:50 EOR
%   B3:4/3  3_EN %
%   B3:5/3  TEST_I3 %
%   B3:5/12  I3_PASS_ZONE %
%   F8:50  I3_TOP_CON_FAILS  "auto stop non pass count top" %

